FUNCTION_BLOCK FB_TestableModuleBase EXTENDS FB_ModuleBase
VAR
	_UpperServiceCtrl : ST_ServiceCtrl;
	_EffectiveServiceCtrl : ST_ServiceCtrl;
	_UpperServiceParam : ST_Chamber1SpinAxisJogParam;
	_EffectiveServiceParam : ST_Chamber1SpinAxisJogParam;
	_ServiceStatus : ST_ServiceStatus;
END_VAR

M_UpdateModule();

METHOD PROTECTED H_RegisterServices
M_RegisterService(
	ServiceId := 1,
	AllowCompositeCall := FALSE,
	UpperCtrl := _UpperServiceCtrl,
	EffectiveCtrl := _EffectiveServiceCtrl,
	UpperParam := _UpperServiceParam,
	EffectiveParam := _EffectiveServiceParam,
	Status := _ServiceStatus);
END_METHOD

METHOD PUBLIC M_SetServiceStatus
VAR_IN_OUT CONSTANT
	Status : ST_ServiceStatus;
END_VAR
_ServiceStatus := Status;
END_METHOD

END_FUNCTION_BLOCK

(* stored: Version 1.1.0.1, ProductVersion 3.1.4026.18
   POU FB_TestableModuleBase: Id {26ed25ca-5582-476d-84bf-1fed652a381d}, SpecialFunc None
   Method H_RegisterServices: Id {5d092d00-e976-450f-a79e-d48e19d42d88}
   Method M_SetServiceStatus: Id {5461878a-0ad3-4d4e-b67a-bcc6acdfcb40} *)
